# EPICS autosave request: iocBoot/sioc-b084-im01/sioc-b084-im01.req
file "lcls2toro.req" AREA=GUNB,POS=360
